FUNCTION FC_InitAlarmTexts : BOOL
VAR_INPUT
END_VAR
VAR
END_VAR

HMI_Texts.AlarmTexts[EAlarms.none] := 'unspecified';
HMI_Texts.AlarmTexts[EAlarms.not_initialized] := 'the component is not initialized yet';
HMI_Texts.AlarmTexts[EAlarms.did_execute] := 'the component executed';
HMI_Texts.AlarmTexts[EAlarms.did_shutdown] := 'the system shut down';

HMI_Texts.AlarmTexts[ESpecialAlarmIds.recovery_request] := 'a recovery was requested';
HMI_Texts.AlarmTexts[ESpecialAlarmIds.definition_request] := 'a definition was requested';

END_FUNCTION

(* stored: Version 1.1.0.1, ProductVersion 3.1.4024.12
   POU FC_InitAlarmTexts: Id {1b864caa-f61e-468a-b82d-180583ccea99}, SpecialFunc None *)
